(*PController:
Implements a simple state feedback law with a 3x3 control gain matrix 'K', 
a translation speed limit 'vtrans_max' (x- and y-axis) and a rotational speed 
limit 'vrot_max'.
*)
FUNCTION_BLOCK PController
VAR_INPUT
	xRobotPose: 		RobotPoseSimple; 				//current pose
	xRobotPoseRef: 		RobotPoseSimple; 				//reference pose
	xRobotvelRef: 		RobotPoseSimple;				//reference velocity
	enable:				BOOL 			:= FALSE;
END_VAR

VAR_OUTPUT
	//control outputs
	vXrobot:			LREAL;
	vYrobot:			LREAL;
	omegaRobot:			LREAL;
	reachedReference:	BOOL;
END_VAR

VAR
	//static control parameters
	K: ARRAY [0..2,0..2] OF LREAL := ControlParameters.controllerK;
	poseError: RobotPoseSimple;
	vtrans_max: LREAL := ControlParameters.vtrans_max;
	vrot_max: LREAL   := ControlParameters.vrot_max; //vTheta
	u: ARRAY[0..2] OF LREAL;
	i: INT;
	accuracyXY: LREAL := ControlParameters.accuracyXY;
	accuracyTheta: LREAL := ControlParameters.accuracyTheta;
END_VAR



//1.) calculate pose errors
poseError.x 	:= xRobotPoseRef.x 		- xRobotPose.x;
poseError.y 	:= xRobotPoseRef.y 		- xRobotPose.y;
poseError.theta := xRobotPoseRef.theta 	- xRobotPose.theta;

reachedReference := (ABS(poseError.x) < accuracyXY) AND (ABS(poseError.y) < accuracyXY) AND (ABS(poseError.theta) < accuracyTheta);

//2.) apply gain on errors
FOR i := 0 TO 2 DO
	u[i] := K[0,i] * poseError.x + K[1,i] * poseError.y + K[2,i] * poseError.theta;
END_FOR;

//3.) apply saturation
FOR i := 0 TO 1 DO
	IF u[i] > vtrans_max THEN
		u[i] := vtrans_max;
	ELSIF u[i] < -vtrans_max THEN
		u[i] := -vtrans_max;
	END_IF
END_FOR

IF u[2] > vrot_max THEN
	u[2] := vrot_max;
ELSIF u[2] < -vrot_max THEN
	u[2] := -vrot_max;
END_IF

//4.) set control outputs
IF enable THEN
	vXrobot 	:= (u[0] + xRobotvelRef.x);
	vYrobot 	:= (u[1] + xRobotvelRef.y);
	omegaRobot	:= (u[2] + xRobotvelRef.theta);
ELSE
	vXrobot 	:= 0;
	vYrobot 	:= 0;
	omegaRobot  := 0;
END_IF

METHOD reset : BOOL
VAR_INPUT
END_VAR
reachedReference := FALSE;
reset := TRUE;
END_METHOD

END_FUNCTION_BLOCK

(* stored: Version 1.1.0.1, ProductVersion 3.1.4024.11
   POU PController: Id {b6b00111-b334-4516-8a6e-fa6dcb5c765f}, SpecialFunc None
   Method reset: Id {abf3cfa0-3136-4152-8add-0d4168a8fd70} *)
